ABB RAPID module: Wizard.modx

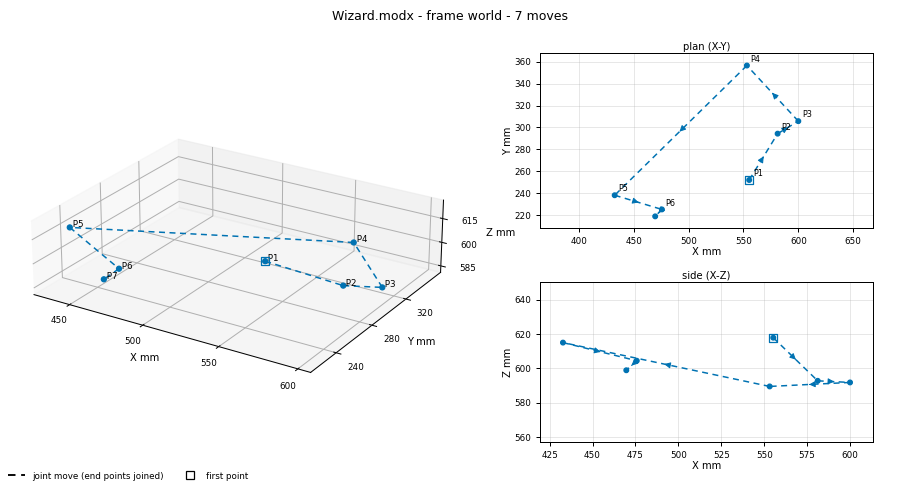
[picture p0: tool path of Wizard.modx in frame world, 7 of 7 moves have a stored position in this frame; points joined in program order, loops and branches not executed]
MODULE Wizard
PERS robtarget O1:=[[356.637451171875, 161.037048339844, 513.128356933594], [0.0388496816158295, -0.776131391525269, -0.358248889446259, -0.517463564872742], [0, 1, 0, 1], [9000000000, 9000000000, 9000000000, 9000000000, 9000000000, 9000000000]];
PERS robtarget O2:=[[356.619445800781, 121.282089233398, 484.093872070313], [0.00313940364867449, -0.806082367897034, -0.327470064163208, -0.492934823036194], [0, 1, 0, 1], [9000000000, 9000000000, 9000000000, 9000000000, 9000000000, 9000000000]];
PERS robtarget O3:=[[399.640594482422, 143.169784545898, 468.373107910156], [0.00769960461184382, 0.794183015823364, 0.382436096668243, 0.472182840108871], [0, 1, 0, 1], [9000000000, 9000000000, 9000000000, 9000000000, 9000000000, 9000000000]];
PERS robtarget O4:=[[436.398681640625, 185.750854492188, 440.245086669922], [0.083333015441895, -0.836603939533234, -0.298512071371078, -0.451707899570465], [0, 1, 0, 1], [9000000000, 9000000000, 9000000000, 9000000000, 9000000000, 9000000000]];
PERS robtarget O5:=[[384.975860595703, 184.290008544922, 436.962097167969], [0.130016103386879, -0.904695689678192, -0.099378101527691, -0.393377006053925], [0, 1, 0, 1], [9000000000, 9000000000, 9000000000, 9000000000, 9000000000, 9000000000]];
PERS robtarget P1:=[[555.272094726563, 252.178009033203, 617.894104003906], [0.081425286829472, 0.61410117149353, -0.783669710159302, -0.0459511838853359], [0, 0, -1, 0], [9000000000, 9000000000, 9000000000, 9000000000, 9000000000, 9000000000]];
PERS robtarget P2:=[[581.155456542969, 294.388061523438, 592.781372070313], [0.188104867935181, 0.633526146411896, -0.750378608703613, 0.0138965677469969], [0, -1, -1, 0], [9000000000, 9000000000, 9000000000, 9000000000, 9000000000, 9000000000]];
PERS robtarget P3:=[[600.000305175781, 305.776336669922, 591.8310546875], [0.121595151722431, 0.64362096786499, -0.755053102970123, 0.0293502137064934], [0, -1, -1, 0], [9000000000, 9000000000, 9000000000, 9000000000, 9000000000, 9000000000]];
PERS robtarget P4:=[[553.178527832031, 356.432434082031, 589.507019042969], [0.16638009250164, 0.676077246665955, -0.716881811618805, 0.0363007448613644], [0, -1, -1, 0], [9000000000, 9000000000, 9000000000, 9000000000, 9000000000, 9000000000]];
PERS robtarget P5:=[[432.768585205078, 238.302230834961, 615.04248046875], [0.0402561873197556, -0.661645650863647, 0.747375845909119, -0.0450976602733135], [0, -1, -1, 0], [9000000000, 9000000000, 9000000000, 9000000000, 9000000000, 9000000000]];
PERS robtarget P6:=[[475.761413574219, 225.393676757813, 604.477722167969], [0.0422640293836594, -0.645888447761536, 0.75911670923233, -0.06916418671608], [0, -1, -1, 0], [9000000000, 9000000000, 9000000000, 9000000000, 9000000000, 9000000000]];
PERS robtarget P7:=[[469.6630859375, 219.079544067383, 598.929931640625], [0.066877692937851, -0.600106239318848, 0.795571863651276, 0.049651961773634], [0, 0, -1, 0], [9000000000, 9000000000, 9000000000, 9000000000, 9000000000, 9000000000]];
	PROC main()
MoveJ P1, v1000, fine, tool0;
MoveJ P2, v1000, fine, tool0;
MoveJ P3, v1000, fine, tool0;
MoveJ P4, v1000, fine, tool0;
MoveJ P5, v1000, fine, tool0;
MoveJ P6, v1000, fine, tool0;
MoveJ P7, v1000, fine, tool0;
	ENDPROC
ENDMODULE
